Yaskawa INFORM job: P_Y_MP.JBI

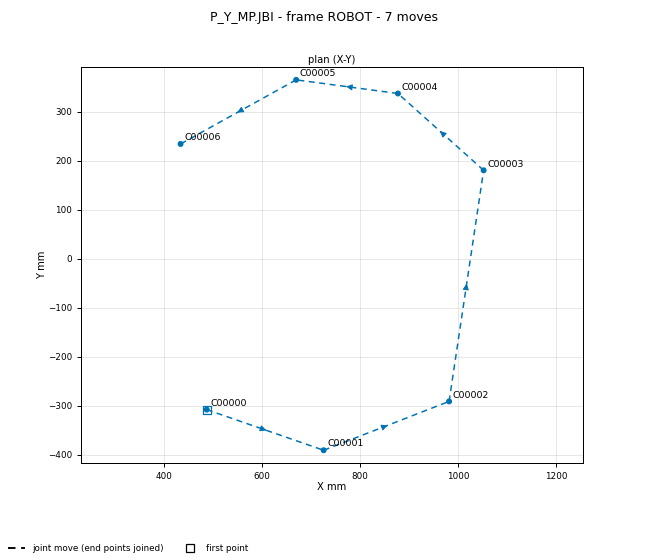
[picture p0: tool path of P_Y_MP.JBI in frame ROBOT, 7 of 7 moves have a stored position in this frame; points joined in program order, loops and branches not executed]
/JOB
//NAME P_Y_MP
///FOLDERNAME INNE
//POS
///NPOS 7,7,7,0,0,0
///TOOL 0
///POSTYPE ROBOT
///RECTAN
///RCONF 0,0,0,0,0,0,0,0,0,0,0,0,0,0,0,0,0,0,0,0,0,0,0,0
C00000=487.677,-308.086,-2138.818,-0.0017,-0.0020,-179.9932
C00001=726.249,-390.964,-2138.479,0.0106,-0.0072,-179.9960
C00002=982.219,-291.307,-2138.442,0.0092,-0.0050,-179.9944
C00003=1052.708,180.254,-2138.006,0.0105,-0.0096,-179.9956
C00004=877.858,336.995,-2138.492,0.0122,-0.0093,179.9989
C00005=670.125,364.845,-2138.389,0.0110,-0.0088,-179.9961
C00006=434.276,234.066,-2138.725,0.0102,-0.0105,-179.9939
BC00000=650.660,6920.928,1262.142
BC00001=650.660,6920.928,1262.142
BC00002=650.660,6920.928,1262.142
BC00003=650.660,6920.928,1262.142
BC00004=650.660,6920.928,1262.142
BC00005=650.660,6920.928,1262.142
BC00006=650.660,6920.928,1262.142
///POSTYPE PULSE
///PULSE
EC00000=0,0
EC00001=0,239555
EC00002=0,501510
EC00003=0,982190
EC00004=0,1204752
EC00005=0,1402700
EC00006=0,1659361
//INST
///DATE 2023/10/04 15:13
///ATTR SC,RW,RJ
////FRAME ROBOT
///GROUP1 RB1,BS1
///GROUP2 ST1
NOP
MOVJ C00000 BC00000 VJ=0.78  +MOVJ EC00000 VJ=0.78
MOVJ C00001 BC00001 VJ=0.78  +MOVJ EC00001 VJ=0.78
MOVJ C00002 BC00002 VJ=0.78  +MOVJ EC00002 VJ=0.78
MOVJ C00003 BC00003 VJ=0.78  +MOVJ EC00003 VJ=0.78
MOVJ C00004 BC00004 VJ=0.78  +MOVJ EC00004 VJ=0.78
MOVJ C00005 BC00005 VJ=0.78  +MOVJ EC00005 VJ=0.78
MOVJ C00006 BC00006 VJ=0.78  +MOVJ EC00006 VJ=0.78
END
